Yaskawa INFORM job: CAL_MINI_STANDARD.JBI

/JOB
//NAME CAL_MINI_STANDARD
//POS
///NPOS 4,0,0,0,0,0
///TOOL 0
///POSTYPE PULSE
///PULSE
C00000=0,-75310,1200,0,-127658,-70
C00001=0,-75310,1200,0,-127658,-70
C00002=45000,-75310,1200,0,-127658,-70
C00003=100,-80000,5000,0,-100000,200
//INST
///DATE 2026/08/22 12:00
///ATTR SC,RW
///GROUP1 RB1
NOP
MSG "STD CAL — Phase A PULSE"
' Confirm cell clear, then CONTINUE
PAUSE
' CALSTEP:home
MSG "STEP_HOME"
' STEP_HOME
' PHASE A — PULSE (standard / pulse job)
' Home / safe pose (anchor)
PAUSE
MOVL C00001 V=50.0
' CALSTEP:uf2_rorg
MSG "STEP_UF2_RORG"
' STEP_UF2_RORG
' UF#2 S1 — RORG (origin)
PAUSE
MOVL C00003 V=50.0
' CALSTEP:joint_limit_S_plus
MSG "STEP_S_PLUS"
' STEP_S_PLUS
' S+ safe limit from home
PAUSE
MOVL C00002 V=50.0
MSG "STD CAL DONE — switch to RELATIVE"
END
